// TIA Portal V20 export
DATA_BLOCK "DataTakeOver_DB"   // DB302
// stored: AutoNumber false, InstanceOfName DataTakeOver, InstanceOfType FB
"DataTakeOver"
   // VAR
   //    Var { ExternalAccessible := 'False'; ExternalVisible := 'False'; ExternalWritable := 'False'} : "TypeVar";
   // END_VAR
BEGIN
END_DATA_BLOCK
